Fanuc KAREL source: kd00040.KL

-- PROVISIONAL review KL for V770-1; original PC SHA256 da77a712f05a516d3542d4182a1f705e67447845cd871ef2f72242b5170aaf6e
-- Incomplete behavior may be omitted. Consult companion uncertainty JSON. Do not deploy.
PROGRAM KD00040
%NOLOCKGROUP
BEGIN
  -- UNRESOLVED_PC offsets 5-26; opcodes AD,32,22,9B,9B,9C,9C,37,2C
  -- UNRESOLVED_PC offsets 31-35; opcodes 7F
END KD00040
